// TIA Portal V15.1 export
// export: Created 2024-05-17T05:38:22.6170331Z, ExportSetting WithDefaults, DisplayName Totally Integrated Automation Portal, DisplayVersion V15.1 Update 5, DisplayName TIA Portal Openness, DisplayVersion V15.1 Update 5, DisplayName SINAMICS Startdrive Advanced, DisplayVersion V15.1, DisplayName G130, G150, S120, S150, SINAMICS MV, S210, DisplayVersion V15.1, DisplayName G110M, G120, G120C, G120D, G120P, DisplayVersion V15.1, DisplayName STEP 7 Professional, DisplayVersion V15.1 Update 5, DisplayName STEP 7 Safety, DisplayVersion V15.1, DisplayName WinCC Professional, DisplayVersion V15.1 Update 5, DisplayName SIMATIC Visualization Architect, DisplayVersion V15.1
DATA_BLOCK "_209230ZM01"   // DB400
{ S7_Optimized_Access := 'FALSE' }
AUTHOR : VCG
VERSION : 0.1
// stored: AutoNumber false, DBAccessibleFromOPCUA true, IsOnlyStoredInLoadMemory false, IsWriteProtectedInAS false
   VAR RETAIN
      AC_209230CA21M4SG1 { ExternalAccessible := 'False'; ExternalVisible := 'False'; ExternalWritable := 'False'} : Bool;   // Detection Buffer first leg full NOK
      AC_209230CA21M4SG3 { ExternalAccessible := 'False'; ExternalVisible := 'False'; ExternalWritable := 'False'} : Bool;   // Detection OK to close Holdback NOK
      AC_209230CA21M4SG4 { ExternalAccessible := 'False'; ExternalVisible := 'False'; ExternalWritable := 'False'} : Bool;   // Detection Buffer second leg full NOK
      AC_209230CA21M4SG9 { ExternalAccessible := 'False'; ExternalVisible := 'False'; ExternalWritable := 'False'} : Bool;   // Detection OK to close Holdback NOK
      AC_BodyCounterConv1 { ExternalAccessible := 'False'; ExternalVisible := 'False'; ExternalWritable := 'False'} : Bool;   // Body Counter below 0 or above MAX
      AlarmA { ExternalAccessible := 'False'; ExternalVisible := 'False'; ExternalWritable := 'False'} : Bool;   // Summary Alarm A
      AlarmB { ExternalAccessible := 'False'; ExternalVisible := 'False'; ExternalWritable := 'False'} : Bool;   // Summary Alarm B
      AlarmC { ExternalAccessible := 'False'; ExternalVisible := 'False'; ExternalWritable := 'False'} : Bool;   // Summary Alarm C
      AlarmD { ExternalAccessible := 'False'; ExternalVisible := 'False'; ExternalWritable := 'False'} : Bool;   // Summary Alarm D
      AlarmABCondition { ExternalAccessible := 'False'; ExternalVisible := 'False'; ExternalWritable := 'False'} : Bool;   // Alarm AB condition
      H_Anim : Word;   // Animation
      H_DBnr : Int;   // DB number
      H_HMICmd : Word;   // HMI Command
      H_OrdersIAnim : DWord;   // HMI Animation of the icon
      H_DataHandlingIAnim : Word;   // HMI Animation of the icon
      H_209230CA21M4SG1IAnim : DWord;   // HMI Animation of the icon
      H_209230CA21M4SG2IAnim : DWord;   // HMI Animation of the icon
      H_209230CA21M4SG3IAnim : DWord;   // HMI Animation of the icon
      H_209230CA21M4SG4IAnim : DWord;   // HMI Animation of the icon
      H_209230CA21M4SG5IAnim : DWord;   // HMI Animation of the icon
      H_209230CA21M4SG9IAnim : DWord;   // HMI Animation of the icon
      H_HMI : Struct   // Icon Animation
         BodyCounter : "H_HMI";   // HMI Animation of the icon
         AndonReq : "H_HMI";   // HMI Animation of the icon
         "209230CHB21" : "H_HMI";   // HMI Animation of the icon
         "209230CHB22" : "H_HMI";   // HMI Animation of the icon
         "209230CA21" : "H_HMI";   // HMI Animation of the icon
         "209230CR22" : "H_HMI";   // HMI Animation of the icon
         "209230CA21M4BufferFull" : "H_HMI";   // HMI Animation of the icon
      END_STRUCT;
      H : Struct   // Animation
         BodyCounter : "H_GBBodyCounter";   // HMI Animation
         AndonReq : "H_AndonReqVCG";   // HMI Animation
         "209230CHB21" : "H_GBMovUnit2Pos2W2S-MoviFitFCPN";   // HMI Animation
         "209230CHB22" : "H_GBMovUnit2Pos2W2S-MoviFitFCPN";   // HMI Animation
         "209230CA21" : "H_GBChain2W1S-MoviFitFCPN";   // HMI Animation
         "209230CR22" : "H_GBRoller2W2S-MoviFitFCPN";   // HMI Animation
         "209230CA21M4BufferFull" : "H_ConditionDelay";   // HMI Animation
      END_STRUCT;
      H_308220ZM01IAnim : Word;   // 308220ZM01: For animation of icon
      H_212DIAnim : Word;   // 212D: For animation of icon
      H_209230CA21FreeSpace : DInt;   // 209230CA21: Free space
      "209230CHB21" { ExternalAccessible := 'False'; ExternalVisible := 'False'; ExternalWritable := 'False'} : "MovUnit";   // HoldBack
      "209230CHB22" { ExternalAccessible := 'False'; ExternalVisible := 'False'; ExternalWritable := 'False'} : "MovUnit";   // HoldBack
      "209230CA21" { ExternalAccessible := 'False'; ExternalVisible := 'False'; ExternalWritable := 'False'} : "Conveyor";   // Roller
      "209230CR22" { ExternalAccessible := 'False'; ExternalVisible := 'False'; ExternalWritable := 'False'} : "Conveyor";   // Roller
      Mode { ExternalAccessible := 'False'; ExternalVisible := 'False'; ExternalWritable := 'False'} : "AlarmBits";   // Mode Alarm Bits / Mode: Summary Alarm A
      Orders { ExternalAccessible := 'False'; ExternalVisible := 'False'; ExternalWritable := 'False'} : "AlarmBits";   // Orders Alarm Bits
      DataHandling { ExternalAccessible := 'False'; ExternalVisible := 'False'; ExternalWritable := 'False'} : "AlarmBits";   // DataHandling Alarm Bits
      BodyCounter { ExternalAccessible := 'False'; ExternalVisible := 'False'; ExternalWritable := 'False'} : "BodyCounter";   // Body Counter
      AndonStatus { ExternalAccessible := 'False'; ExternalVisible := 'False'; ExternalWritable := 'False'} : "AndonStatusVCG";   // Andon - Status
      AndonDataExchange { ExternalAccessible := 'False'; ExternalVisible := 'False'; ExternalWritable := 'False'} : "AndonDataExchangeVCG";   // Andon - Data Exchange
      HomePosition { ExternalAccessible := 'False'; ExternalVisible := 'False'; ExternalWritable := 'False'} : Bool;   // Home position
      EmptyStnReached { ExternalAccessible := 'False'; ExternalVisible := 'False'; ExternalWritable := 'False'} : Bool;   // Empty Station is Reached
      "230CA21M4SG1CheckOn" { ExternalAccessible := 'False'; ExternalVisible := 'False'; ExternalWritable := 'False'} : Bool;   // Check On Buffer first leg full
      "230CA21M4SG1DetOn" { ExternalAccessible := 'False'; ExternalVisible := 'False'; ExternalWritable := 'False'} : Bool;   // Buffer first leg full
      "230CA21M4SG2DetOn" { ExternalAccessible := 'False'; ExternalVisible := 'False'; ExternalWritable := 'False'} : Bool;   // Holdback Occupied
      "230CA21M4SG3CheckOn" { ExternalAccessible := 'False'; ExternalVisible := 'False'; ExternalWritable := 'False'} : Bool;   // Check On OK to close Holdback
      "230CA21M4SG3DetOn" { ExternalAccessible := 'False'; ExternalVisible := 'False'; ExternalWritable := 'False'} : Bool;   // OK to close Holdback
      "230CA21M4SG4CheckOn" { ExternalAccessible := 'False'; ExternalVisible := 'False'; ExternalWritable := 'False'} : Bool;   // Check On Buffer second leg full
      "230CA21M4SG4DetOn" { ExternalAccessible := 'False'; ExternalVisible := 'False'; ExternalWritable := 'False'} : Bool;   // Buffer second leg full
      "230CA21M4SG5DetOn" { ExternalAccessible := 'False'; ExternalVisible := 'False'; ExternalWritable := 'False'} : Bool;   // Holdback Occupied
      "230CA21M4SG9CheckOn" { ExternalAccessible := 'False'; ExternalVisible := 'False'; ExternalWritable := 'False'} : Bool;   // Check On OK to close Holdback
      "230CA21M4SG9DetOn" { ExternalAccessible := 'False'; ExternalVisible := 'False'; ExternalWritable := 'False'} : Bool;   // OK to close Holdback
      "230CA21M4FreeSpaceActive" { ExternalAccessible := 'False'; ExternalVisible := 'False'; ExternalWritable := 'False'} : Bool;   // HMI command: Free space active
      "230CA21M4FreeSpace" { ExternalAccessible := 'False'; ExternalVisible := 'False'; ExternalWritable := 'False'} : Bool;   // Free space
      "230CA21M4BufferFull" { ExternalAccessible := 'False'; ExternalVisible := 'False'; ExternalWritable := 'False'} : Bool;   // Buffer Full
      Edge { ExternalAccessible := 'False'; ExternalVisible := 'False'; ExternalWritable := 'False'} : Array[1..10] of Bool;   // Edge
   END_VAR
BEGIN
END_DATA_BLOCK
